INTERFACE I_UniversalAxisCA EXTENDS I_UniversalAxis

PROPERTY DirectionCA : Tc3_Mc3Definitions.MC_DIRECTION
GET
END_GET
SET
END_SET
END_PROPERTY

PROPERTY Gap : MC_LREAL
GET
END_GET
SET
END_SET
END_PROPERTY

PROPERTY HaltedCA : REFERENCE TO BOOL
GET
END_GET
END_PROPERTY

METHOD MR_HaltCA : BOOL
VAR_INPUT
END_VAR
END_METHOD

METHOD MR_MoveAbsoluteCA : BOOL
VAR_INPUT
	lrAbsolutePosition : LREAL;
END_VAR
END_METHOD

METHOD MR_MoveRelativeCA : BOOL
VAR_INPUT
	lrRelativeDistance : LREAL;
END_VAR
END_METHOD

PROPERTY StateCA : REFERENCE TO E_AxisStateCA
GET
END_GET
END_PROPERTY

END_INTERFACE

(* stored: Version 1.1.0.1, ProductVersion 3.1.4024.12
   Itf I_UniversalAxisCA: Id {71f2142d-11f6-4578-bf9e-be59a6d688c8}
   Property DirectionCA: Id {40560496-ce00-4387-a16a-793c931ebc35}
   Get Get: Id {467a9772-21ee-4535-9c95-f3f859bbc5b8}
   Set Set: Id {50ae83fc-2b60-4f45-ad0b-d13f7369cad6}
   Property Gap: Id {df199cf0-7e1a-488a-919c-e1632e969ed6}
   Get Get: Id {0c35475f-1734-43d4-ab26-76319bff7474}
   Set Set: Id {8d1c9294-5fed-4deb-8022-1a4e4adcc489}
   Property HaltedCA: Id {fcd41d24-0918-4a2f-8a84-6e033be2404f}
   Get Get: Id {88b14bf8-2bf0-45db-8585-97930d322b70}
   Method MR_HaltCA: Id {28c2dbe2-1869-47a7-9f8c-786e3a147353}
   Method MR_MoveAbsoluteCA: Id {ad9263c4-012e-4621-abe1-e3e191589481}
   Method MR_MoveRelativeCA: Id {aab0e32b-87d0-46a1-9099-b0fd17247068}
   Property StateCA: Id {77a0948c-cca0-42de-85da-2442ae6ea5bf}
   Get Get: Id {7db3c847-997c-499e-87fb-1efbe03e31cf} *)
